Staubli VAL3: OMAC_Hold.pgx

program OMAC_Hold()
  local joint l_jHere
begin
  //OMAC进程:Holding
  _nOmacStat=5
  logMsg("上位机手动操作：暂停")
  _bEndCycle=true
  wait(taskStatus("productionCycle")==-1)
  _bMutexCnvQueue[0]=false
  taskKill("cellManager")
  wait(taskStatus("cellManager")==-1)
  stopMove()
  resetMotion()
  // Move up axis 3
  l_jHere=herej()
  l_jHere.j3=95
  movej(l_jHere,tGripper,mSlow)
  movej(jHome,tGripper,mSlow)
  waitEndMove()
  disablePower()
  dVacuum=false
  wait(isSettled())
  wait(isPowered()==false)
  //OMAC进程:Held
  _nOmacStat=6
  delay(0)
end
